{attribute 'qualified_only'}
{attribute 'strict'}
TYPE E_Message_Battery :
(
	eNoMessage := 0,
	eTooMuchBattery := 1,
	eBatteryError := 2,
	eNoConnectionToBackend := 3
);
END_TYPE

(* stored: Version 1.1.0.1, ProductVersion 3.1.4024.6
   DUT E_Message_Battery: Id {f1b77947-7421-4dbd-9448-ec1657a4c526} *)
